Universal Robots PolyScope program: test_circ_motion.urp

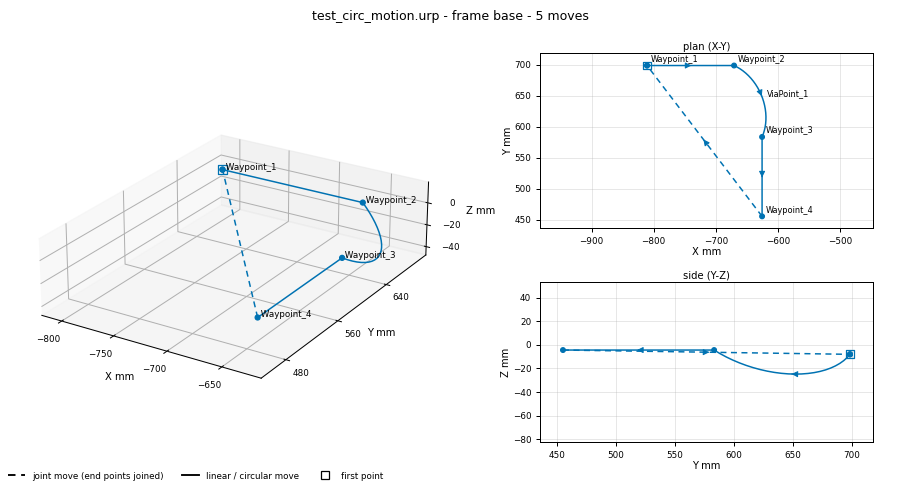
[picture p0: tool path of test_circ_motion.urp in frame base, 5 of 6 moves have a stored position in this frame; points joined in program order, loops and branches not executed]
Program test_circ_motion (installation=default directory=/programs createdIn=5.14.5 lastSavedIn=5.14.5 robotSerialNumber=20236801216)
Calibrated DH parameters: a=[-0.000021, -0.748897, -0.28186, -0.00004, -0.000055, 0]; d=[0.236225, -424.082933, -1564.66872, 1988.95162, 0.159094, 0.153873]; alpha=[1.570844, 0.001002, 0.000337, 1.571488, -1.569996, 0]; deltaTheta=[0, -0.516316, 5.626292, 1.173211, 0.000001, 0]
InitVariablesNode
Robot Program (runOnlyOnce=true)
  MoveJ speed 60 deg/s, acceleration 80 deg/s^2 (useActiveTCP=true) feature=Base
    Waypoint Waypoint_1: TCP in base x=-810.726 y=698.393 z=-8.087 mm, rx=1.5708 ry=0 rz=0 rad; joints [-56.676, -33.897, 84.846, -50.837, -56.733, -0.134] deg; TCP offset x=0 y=0 z=19 mm, rx=0 ry=0 rz=0 rad
  MoveL speed 250 mm/s, acceleration 1200 mm/s^2 (useActiveTCP=true) feature=Base
    Waypoint Waypoint_2: TCP in base x=-670.488 y=698.404 z=-8.079 mm, rx=1.5708 ry=0 rz=0 rad; joints [-62.84, -37.511, 94.354, -56.747, -62.898, -0.118] deg
  MoveP speed 250 mm/s, acceleration 1200 mm/s^2 (blendRadius=0.025 useActiveTCP=true) feature=Base
    CircleMove (OrientationMode=FIXED)
      Waypoint ViaPoint_1: TCP in base x=-623.805 y=643.42 z=-24.462 mm, rx=0.6268 ry=-1.4796 rz=0.656 rad; joints [-69.172, -20.539, 103.252, -262.494, 26.209, 270.871] deg
      Waypoint Waypoint_3: TCP in base x=-625.327 y=583.309 z=-4.461 mm, rx=0 ry=-1.5708 rz=0 rad; joints [-67.863, -22.034, 118.956, 83.161, -22.102, -90.072] deg
  MoveL speed 250 mm/s, acceleration 1200 mm/s^2 (useActiveTCP=true) feature=Base
    Waypoint Waypoint_4: TCP in base x=-625.332 y=455.317 z=-4.463 mm, rx=0 ry=-1.5708 rz=-0.0001 rad; joints [-63.277, -20.477, 126.164, 74.382, -26.692, -90.059] deg
  MoveJ speed 60 deg/s, acceleration 80 deg/s^2 (useActiveTCP=true) feature=Base
    Waypoint Waypoint_1: TCP in base x=-810.726 y=698.393 z=-8.087 mm, rx=1.5708 ry=0 rz=0 rad; joints [-56.676, -33.897, 84.846, -50.837, -56.733, -0.134] deg
